# EPICS autosave request: mrfApp/Db/evr-template-pulse-gen-prescaler-16-bit.inc.req
$(P)$(R)PulseGen@PULSE_GEN_NUM@:Prescaler.VAL
